(* IEC 61131-3 sources: matiec/tests/corpus_attr, 19 files *)

(* ---- attr_before_fb.st ---- *)
{attribute 'label' := 'demo'}
FUNCTION_BLOCK fb
VAR_INPUT i : INT; END_VAR
VAR_OUTPUT o : INT; END_VAR
o := i;
END_FUNCTION_BLOCK

(* ---- attr_in_var_output.st ---- *)
FUNCTION_BLOCK fb
VAR_INPUT i : INT; END_VAR
VAR_OUTPUT
  {attribute 'label' := 'o'}
  o : INT;
END_VAR
o := i;
END_FUNCTION_BLOCK

(* ---- pragma_plain_in_var_output.st ---- *)
FUNCTION_BLOCK fb
VAR_INPUT i : INT; END_VAR
VAR_OUTPUT
  {some_vendor_pragma}
  o : INT;
END_VAR
o := i;
END_FUNCTION_BLOCK

(* ---- attr_before_action.st ---- *)
PROGRAM p
VAR x : BOOL; END_VAR
INITIAL_STEP s0: END_STEP
TRANSITION FROM s0 TO s1 := x; END_TRANSITION
STEP s1: a(N); END_STEP
TRANSITION FROM s1 TO s0 := NOT x; END_TRANSITION
{attribute 'label' := 'a'}
ACTION a: x := FALSE; END_ACTION
END_PROGRAM

(* ---- attr_before_initial_step.st ---- *)
PROGRAM p
VAR x : BOOL; END_VAR
{attribute 'label' := 's0'}
INITIAL_STEP s0: END_STEP
TRANSITION FROM s0 TO s1 := x; END_TRANSITION
STEP s1: a(N); END_STEP
TRANSITION FROM s1 TO s0 := NOT x; END_TRANSITION
ACTION a: x := FALSE; END_ACTION
END_PROGRAM

(* ---- attr_before_step.st ---- *)
PROGRAM p
VAR x : BOOL; END_VAR
INITIAL_STEP s0: END_STEP
TRANSITION FROM s0 TO s1 := x; END_TRANSITION
{attribute 'label' := 's1'}
STEP s1: a(N); END_STEP
TRANSITION FROM s1 TO s0 := NOT x; END_TRANSITION
ACTION a: x := FALSE; END_ACTION
END_PROGRAM

(* ---- attr_before_transition.st ---- *)
PROGRAM p
VAR x : BOOL; END_VAR
INITIAL_STEP s0: END_STEP
{attribute 'label' := 't0'}
TRANSITION FROM s0 TO s1 := x; END_TRANSITION
STEP s1: a(N); END_STEP
TRANSITION FROM s1 TO s0 := NOT x; END_TRANSITION
ACTION a: x := FALSE; END_ACTION
END_PROGRAM

(* ---- attr_before_var_block.st ---- *)
PROGRAM p
{attribute 'label' := 'blk'}
VAR x : INT; END_VAR
x := x + 1;
END_PROGRAM

(* ---- attr_in_and_out_comment.st ---- *)
(* {attribute 'label' := 'c'} *)
{attribute 'label' := 'demo'}
PROGRAM p
VAR
  (* {attribute 'label' := 'c'} *) {attribute 'label' := 'x'}
  x : INT;
END_VAR
x := x + 1;
END_PROGRAM

(* ---- attr_in_body.st ---- *)
PROGRAM p
VAR x : INT; END_VAR
{attribute 'label' := 'stmt'}
x := x + 1;
END_PROGRAM

(* ---- attr_in_comment.st ---- *)
(* {attribute 'label' := 'demo'} *)
PROGRAM p
VAR
  (* {attribute 'label' := 'x'} *)
  x : INT;
END_VAR
x := x + 1;
END_PROGRAM

(* ---- attr_in_var.st ---- *)
PROGRAM p
VAR
  {attribute 'label' := 'x'}
  x : INT;
END_VAR
x := x + 1;
END_PROGRAM

(* ---- attr_in_var_external.st ---- *)
PROGRAM p
VAR_EXTERNAL
  {attribute 'label' := 'g'}
  g : INT;
END_VAR
g := g + 1;
END_PROGRAM

(* ---- attr_multi_field.st ---- *)
{attribute 'label' := 'demo'}
{attribute 'flag'}
{attribute 'pair' := 'k1', 'k2' := 'v2'}
PROGRAM p
VAR
  {attribute 'label' := 'x'} {attribute 'flag'}
  x : INT;
END_VAR
x := x + 1;
END_PROGRAM

(* ---- base_no_attr.st ---- *)
PROGRAM p
VAR x : INT; END_VAR
x := x + 1;
END_PROGRAM

(* ---- base_sfc.st ---- *)
PROGRAM p
VAR x : BOOL; END_VAR
INITIAL_STEP s0: END_STEP
TRANSITION FROM s0 TO s1 := x; END_TRANSITION
STEP s1: a(N); END_STEP
TRANSITION FROM s1 TO s0 := NOT x; END_TRANSITION
ACTION a: x := FALSE; END_ACTION
END_PROGRAM

(* ---- pragma_plain_before_step.st ---- *)
PROGRAM p
VAR x : BOOL; END_VAR
INITIAL_STEP s0: END_STEP
TRANSITION FROM s0 TO s1 := x; END_TRANSITION
{some_vendor_pragma}
STEP s1: END_STEP
TRANSITION FROM s1 TO s0 := NOT x; END_TRANSITION
END_PROGRAM

(* ---- seed_attr_before_program.st ---- *)
{attribute 'label' := 'demo'}
PROGRAM p
VAR x : INT; END_VAR
x := x + 1;
END_PROGRAM

(* ---- seed_attr_in_var_input.st ---- *)
{attribute 'label' := 'demo'}
PROGRAM p
VAR_INPUT
  {attribute 'label' := 'v'}
  v : REAL := 1.0;
END_VAR
VAR x : INT; END_VAR
x := x + 1;
END_PROGRAM
